(* CoDeSys 2.3 export: PLC_PRG.EXP *)

(* POU PLC_PRG, LD *)
PROGRAM PLC_PRG
(*
	 autor; franklin
	 descricao: codigo estruturado com base em um autômato finito determinísco (AFD) para controle de maquina de estados finita
*)

VAR
	botao AT %IX0.0: BOOL;
	S0 AT %MX0.0: BOOL;
	T1: TON;
	A_VERDE AT %QX1.2: BOOL;
	B_VERMELHO AT %QX1.3: BOOL;
	S1 AT %MX0.1: BOOL;
	botao_pulso: R_TRIG;
	A_AMARELO AT %QX1.1: BOOL;
	T2: TON;
	S2 AT %MX0.2: BOOL;
	B_VERDE AT %QX1.5: BOOL;
	S3 AT %MX0.3: BOOL;
	A_VERMELHO AT %QX1.0: BOOL;
	B_AMARELO AT %QX1.4: BOOL;
	T3: TON;
	T4: TON;
END_VAR
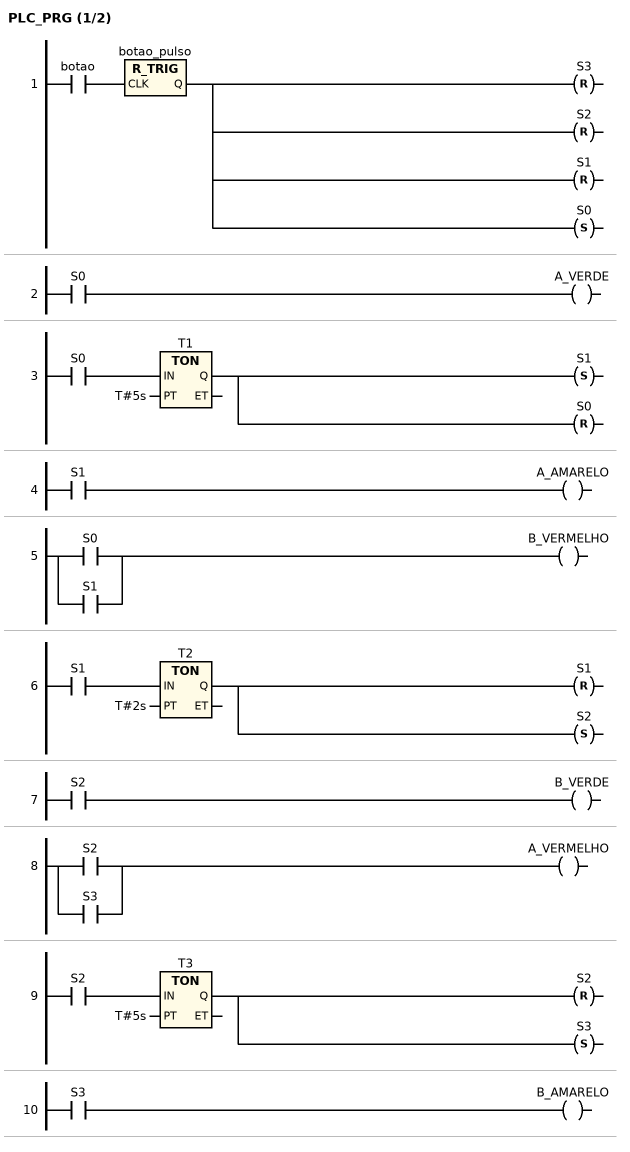
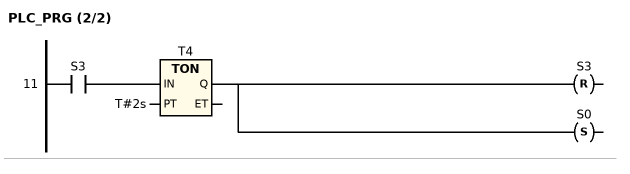
_LD_ (* Ladder Diagram *)
NETWORK 1
	[botao] - botao_pulso:R_TRIG(CLK: *) --- (R S3) (R S2) (R S1) (S S0)
NETWORK 2
	[S0] --- (A_VERDE)
NETWORK 3
	[S0] - T1:TON(IN: *, PT: T#5s) --- (S S1) (R S0)
NETWORK 4
	[S1] --- (A_AMARELO)
NETWORK 5
	{ [S0] | [S1] } --- (B_VERMELHO)
NETWORK 6
	[S1] - T2:TON(IN: *, PT: T#2s) --- (R S1) (S S2)
NETWORK 7
	[S2] --- (B_VERDE)
NETWORK 8
	{ [S2] | [S3] } --- (A_VERMELHO)
NETWORK 9
	[S2] - T3:TON(IN: *, PT: T#5s) --- (R S2) (S S3)
NETWORK 10
	[S3] --- (B_AMARELO)
NETWORK 11
	[S3] - T4:TON(IN: *, PT: T#2s) --- (R S3) (S S0)
_END_LD_
(* the same logic as Structured Text *)
(* Network 1 *)
botao_pulso(CLK := botao);
IF botao_pulso.Q THEN S3 := FALSE; S2 := FALSE; S1 := FALSE; S0 := TRUE; END_IF;
(* Network 2 *)
A_VERDE := S0;
(* Network 3 *)
T1(IN := S0, PT := T#5s);
IF T1.Q THEN S1 := TRUE; S0 := FALSE; END_IF;
(* Network 4 *)
A_AMARELO := S1;
(* Network 5 *)
B_VERMELHO := S0 OR S1;
(* Network 6 *)
T2(IN := S1, PT := T#2s);
IF T2.Q THEN S1 := FALSE; S2 := TRUE; END_IF;
(* Network 7 *)
B_VERDE := S2;
(* Network 8 *)
A_VERMELHO := S2 OR S3;
(* Network 9 *)
T3(IN := S2, PT := T#5s);
IF T3.Q THEN S2 := FALSE; S3 := TRUE; END_IF;
(* Network 10 *)
B_AMARELO := S3;
(* Network 11 *)
T4(IN := S3, PT := T#2s);
IF T4.Q THEN S3 := FALSE; S0 := TRUE; END_IF;
END_PROGRAM
